# EPICS StreamDevice protocol: hp-1-0/proto/E4419B.proto
# HP E4419B Communication Protocol
# Author : Seung-hee Nam
# email : namsh@korea.ac.kr / beyourangel1@gmail.com
# Data : Tuesday, November 15 17:47 KST 2022
# Data format
#       baud rate : 9600
#       parity : None
#       data : 8
#       stop : 1
# Communication procedure
# Transmit Protocol : SCPI
# Terminator : LF

InTerminator = LF;
OutTerminator = LF;
ExtraInput = Ignore;

getIDN {
    out "*IDN?";
    in "%\$1[^\r\n]";
    ExtraInput = Ignore;
}
cmd {
    out "\$1";
}

cmd1 {
    out "\$1 1";
}

setD {
    out "\$1 %d";
    @init { out "\$1?"; in "%d"; }
}
getD {
    out "\$1?";
    in "%d";
    ExtraInput = Ignore;
}

getF
{
    ReplyTimeout = 5000;
    out "\$1?";
    in  "%f";
}
getS
{
    out "\$1?";
    in  "%s";
}

setF
{
    out "\$1 %f";
    @init { getF; }
}

getChA
{
    out "\$1?";
    in "%s";
    ExtraInput = Ignore;
}
